TYPE U_Word :
UNION
	iINT		:INT;
	uiUINT		:UINT;
	
	wWORD		:WORD;
END_UNION
END_TYPE

(* stored: Version 1.1.0.1, ProductVersion 3.1.4026.12
   DUT U_Word: Id {fdeaf71b-b56b-4203-8441-a49b3caec158} *)
